// TIA Portal project "Water Control" (V16)

(* hardware
DEVICE "HMI_1"  TP1500 Comfort Portrait
   slot 0: "HMI_1"  TP1500 Comfort Portrait  6AV2 124-0QC02-0AX0  16.0.0.0
   slot 1: "HMI_RT_1"  TP1500 Comfort Portrait  6AV2 124-0QC02-0AX0  16.0.0.0
   slot 5: "HMI_1.IE_CP_1"  PROFINET Interface  16.0.0.0
      slot 1: "PROFINET Interface_1"  PROFINET Interface
         slot 1: "Port_1"  Port
         slot 2: "Port_2"  Port
   slot 6: "HMI_1.IE_CP_2"  PROFINET Interface  16.0.0.0
      slot 1: "PROFINET Interface_GBit"  PROFINET Interface
         slot 1: "Port_1"  Port
   slot 7: "HMI_1.MPI/DP_CP_1"  MPI/DP Interface  16.0.0.0
DEVICE "S71500/ET200MP station_1"  S7-1500 station
   slot 0: "Rail_0"  Rack  6ES7 590-1***0-0AA0
   slot 1: "PLC_1"  CPU 1511-1 PN  6ES7 511-1AK02-0AB0  V2.8
      slot 3: "CPU display_1"  6ES7591-1AA00-0AA0
      slot 32768: "PROFINET interface_1"  X1
         slot 32769: "Port_1"  X1 P1
         slot 32770: "Port_2"  X1 P2
      slot 34817: "Virtual CP interface port_1"  Virtual CP interface port  Virtual CP interface port
*)

// ===== PLC "PLC_1"  CPU 1511-1 PN =====

VAR_GLOBAL   // PLC tag table "Default tag table"
   "Min. Water Level" AT %M0.0 : Bool;
   "Lower Water Level" AT %M0.1 : Bool;
   "Upper Water Level" AT %M0.2 : Bool;
   "Max. Water Level" AT %M0.3 : Bool;
   "Heating" AT %M1.1 : Bool;
   "Inlet Valve Slow" AT %M1.2 : Bool;
   "Inlet Valve Fast" AT %M1.3 : Bool;
   "Oulet Valve" AT %M1.4 : Bool;
   "Water Level" AT %M0.4 : Bool;
   "PTRIG1" AT %M0.5 : Bool;
   "PTRIG2" AT %M0.6 : Bool;
   "PTRIG3" AT %M0.7 : Bool;
   "PTRIG4" AT %M1.0 : Bool;
   "PTRIG5" AT %M1.5 : Bool;
   "Start" AT %M2.0 : Bool;
   "PTRIG6" AT %M1.6 : Bool;
   "Min Sensör arızalı" AT %M1.7 : Bool;
   "RESET" AT %M2.1 : Bool;
END_VAR

DATA_BLOCK "Sıcaklık Bilgileri"   // DB1
{ S7_Optimized_Access := 'TRUE' }
VERSION : 0.1
   VAR
      "Temp. Min Set" : Real;
      "Temp. Max Set" : Real;
      "Temp.Act Value" : Int;
      "Temp Min" : Bool;
      Heating : Bool;
      "Temp Max" : Bool;
   END_VAR
BEGIN
END_DATA_BLOCK

ORGANIZATION_BLOCK "Main"   // OB1, LAD, ProgramCycle
TITLE = "Main Program Sweep (Cycle)"
{ S7_Optimized_Access := 'TRUE' }
VERSION : 0.1
   VAR_INPUT
      Initial_Call : Bool;   // Initial call of this OB
      Remanence : Bool;   // =True, if remanent data are available
   END_VAR
   VAR_TEMP   // added for the SCL form of the ladder/FBD networks
      _w1 : Bool;
      _w2 : Bool;
      _w3 : Bool;
      _w4 : Bool;
      _w5 : Bool;
      _w6 : Bool;
   END_VAR
BEGIN

REGION Network 1: Min Max Temp info
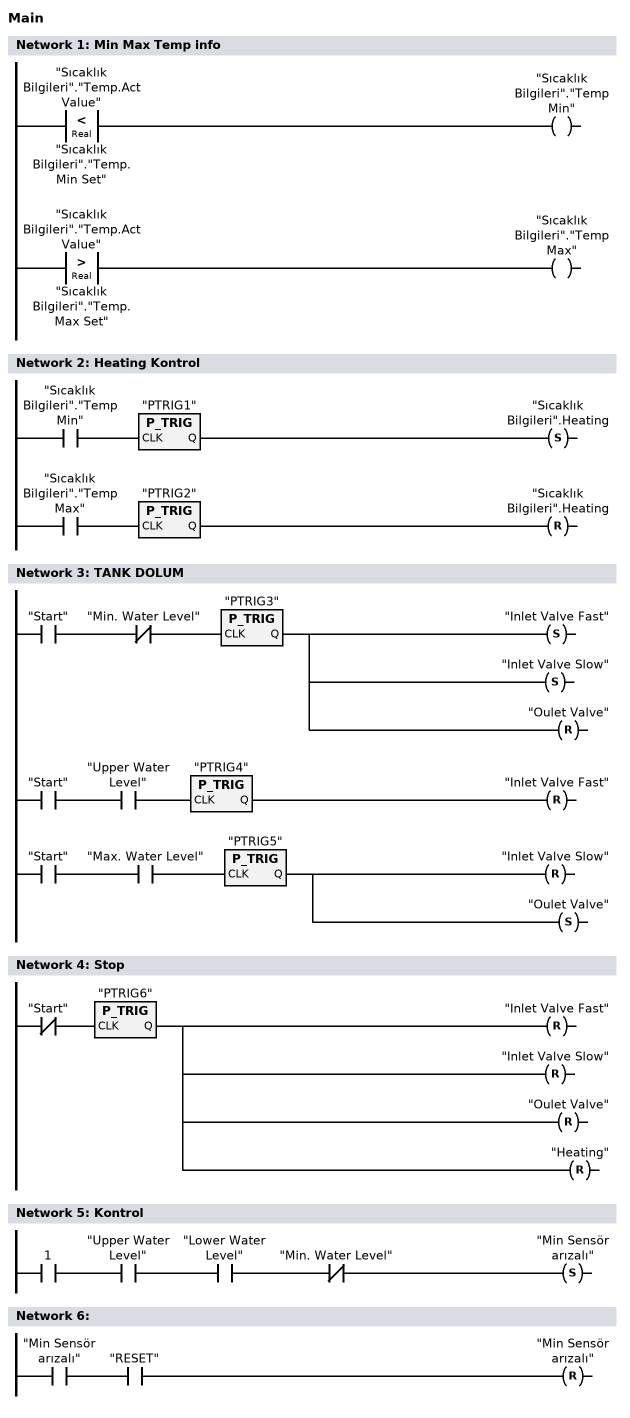
   RUNG wire#powerrail
      { S7_Templates := "SrcType := Real" } LT_Contact(in1 := "Sıcaklık Bilgileri"."Temp.Act Value", in2 := "Sıcaklık Bilgileri"."Temp. Min Set")
      Coil( "Sıcaklık Bilgileri"."Temp Min" )
   END_RUNG
   RUNG wire#powerrail
      { S7_Templates := "SrcType := Real" } GT_Contact(in1 := "Sıcaklık Bilgileri"."Temp.Act Value", in2 := "Sıcaklık Bilgileri"."Temp. Max Set")
      Coil( "Sıcaklık Bilgileri"."Temp Max" )
   END_RUNG
   // the same network as SCL:
   "Sıcaklık Bilgileri"."Temp Min" := "Sıcaklık Bilgileri"."Temp.Act Value" < "Sıcaklık Bilgileri"."Temp. Min Set";
   "Sıcaklık Bilgileri"."Temp Max" := "Sıcaklık Bilgileri"."Temp.Act Value" > "Sıcaklık Bilgileri"."Temp. Max Set";
END_REGION

REGION Network 2: Heating Kontrol
   RUNG wire#powerrail
      Contact( "Sıcaklık Bilgileri"."Temp Min" )
      P_Trig( "PTRIG1" )
      S_Coil( "Sıcaklık Bilgileri".Heating )
   END_RUNG
   RUNG wire#powerrail
      Contact( "Sıcaklık Bilgileri"."Temp Max" )
      P_Trig( "PTRIG2" )
      R_Coil( "Sıcaklık Bilgileri".Heating )
   END_RUNG
   // the same network as SCL:
   #_w1 := "Sıcaklık Bilgileri"."Temp Min" AND NOT "PTRIG1";   // rising edge
   "PTRIG1" := "Sıcaklık Bilgileri"."Temp Min";
   IF #_w1 THEN "Sıcaklık Bilgileri".Heating := TRUE; END_IF;
   #_w2 := "Sıcaklık Bilgileri"."Temp Max" AND NOT "PTRIG2";   // rising edge
   "PTRIG2" := "Sıcaklık Bilgileri"."Temp Max";
   IF #_w2 THEN "Sıcaklık Bilgileri".Heating := FALSE; END_IF;
END_REGION

REGION Network 3: TANK DOLUM
   RUNG wire#powerrail
      Contact( "Start" )
      I_Contact( "Min. Water Level" )
      P_Trig( "PTRIG3" )
      wire#w1
      S_Coil( "Inlet Valve Fast" )
   END_RUNG
   RUNG wire#w1
      S_Coil( "Inlet Valve Slow" )
   END_RUNG
   RUNG wire#w1
      R_Coil( "Oulet Valve" )
   END_RUNG
   RUNG wire#powerrail
      Contact( "Start" )
      Contact( "Upper Water Level" )
      P_Trig( "PTRIG4" )
      R_Coil( "Inlet Valve Fast" )
   END_RUNG
   RUNG wire#powerrail
      Contact( "Start" )
      Contact( "Max. Water Level" )
      P_Trig( "PTRIG5" )
      wire#w2
      R_Coil( "Inlet Valve Slow" )
   END_RUNG
   RUNG wire#w2
      S_Coil( "Oulet Valve" )
   END_RUNG
   // the same network as SCL:
   #_w1 := "Start" AND NOT "Min. Water Level";
   #_w2 := #_w1 AND NOT "PTRIG3";   // rising edge
   "PTRIG3" := #_w1;
   IF #_w2 THEN
       "Inlet Valve Fast" := TRUE;
       "Inlet Valve Slow" := TRUE;
       "Oulet Valve" := FALSE;
   END_IF;
   #_w3 := "Start" AND "Upper Water Level";
   #_w4 := #_w3 AND NOT "PTRIG4";   // rising edge
   "PTRIG4" := #_w3;
   IF #_w4 THEN "Inlet Valve Fast" := FALSE; END_IF;
   #_w5 := "Start" AND "Max. Water Level";
   #_w6 := #_w5 AND NOT "PTRIG5";   // rising edge
   "PTRIG5" := #_w5;
   IF #_w6 THEN
       "Inlet Valve Slow" := FALSE;
       "Oulet Valve" := TRUE;
   END_IF;
END_REGION

REGION Network 4: Stop
   RUNG wire#powerrail
      I_Contact( "Start" )
      P_Trig( "PTRIG6" )
      wire#w1
      R_Coil( "Inlet Valve Fast" )
   END_RUNG
   RUNG wire#w1
      R_Coil( "Inlet Valve Slow" )
   END_RUNG
   RUNG wire#w1
      R_Coil( "Oulet Valve" )
   END_RUNG
   RUNG wire#w1
      R_Coil( "Heating" )
   END_RUNG
   // the same network as SCL:
   #_w1 := NOT "Start" AND NOT "PTRIG6";   // rising edge
   "PTRIG6" := NOT "Start";
   IF #_w1 THEN
       "Inlet Valve Fast" := FALSE;
       "Inlet Valve Slow" := FALSE;
       "Oulet Valve" := FALSE;
       "Heating" := FALSE;
   END_IF;
END_REGION

REGION Network 5: Kontrol
   RUNG wire#powerrail
      Contact( 1 )
      Contact( "Upper Water Level" )
      Contact( "Lower Water Level" )
      I_Contact( "Min. Water Level" )
      S_Coil( "Min Sensör arızalı" )
   END_RUNG
   // the same network as SCL:
   IF 1 AND "Upper Water Level" AND "Lower Water Level" AND NOT "Min. Water Level" THEN
       "Min Sensör arızalı" := TRUE;
   END_IF;
END_REGION

REGION Network 6
   RUNG wire#powerrail
      Contact( "Min Sensör arızalı" )
      Contact( "RESET" )
      R_Coil( "Min Sensör arızalı" )
   END_RUNG
   // the same network as SCL:
   IF "Min Sensör arızalı" AND "RESET" THEN "Min Sensör arızalı" := FALSE; END_IF;
END_REGION
END_ORGANIZATION_BLOCK

(* ===== HMI "HMI_RT_1" =====
system functions are stored by id; their names below are inferred from use
connection "HMI_Connection_3": ETHERNET, S7_1500_OMS

HMI tags "Default tag table"
   "Tag_ScreenNumber" : UInt, internal
   "Sıcaklık Bilgileri_Temp. Min Set" : Real = PLC "Sıcaklık Bilgileri"."Temp. Min Set", 1 s
   "Sıcaklık Bilgileri_Temp. Max Set" : Real = PLC "Sıcaklık Bilgileri"."Temp. Max Set", 1 s
   "Inlet Valve Fast" : Bool = PLC "Inlet Valve Fast" AT %M1.3, 1 s
   "Inlet Valve Slow" : Bool = PLC "Inlet Valve Slow" AT %M1.2, 1 s
   "Oulet Valve" : Bool = PLC "Oulet Valve" AT %M1.4, 1 s
   "Sıcaklık Bilgileri_Temp Min" : Bool = PLC "Sıcaklık Bilgileri"."Temp Min", 1 s
   "Sıcaklık Bilgileri_Temp Max" : Bool = PLC "Sıcaklık Bilgileri"."Temp Max", 1 s
   "Min. Water Level" : Bool = PLC "Min. Water Level" AT %M0.0, 1 s
   "Upper Water Level" : Bool = PLC "Upper Water Level" AT %M0.2, 1 s
   "Max. Water Level" : Bool = PLC "Max. Water Level" AT %M0.3, 1 s
   "Lower Water Level" : Bool = PLC "Lower Water Level" AT %M0.1, 1 s
   "Sıcaklık Bilgileri_Temp.Act Value" : Int = PLC "Sıcaklık Bilgileri"."Temp.Act Value", 1 s
   "Sıcaklık Bilgileri_Heating" : Bool = PLC "Sıcaklık Bilgileri".Heating, 1 s
   "Start" : Bool = PLC Start AT %M2.0, 1 s
   "RESET" : Bool = PLC RESET AT %M2.1, 1 s
   "Min Sensör arızalı" : Bool = PLC "Min Sensör arızalı" AT %M1.7, 1 s

screen "Root screen" 800x1220, template "Template_1"
   on GenerateScreen: SetTag("Tag_ScreenNumber", 1)
   IOField "I/O field_1" at 265,163 size 138x37; FormatPattern 9999.9
      ProcessValue <- "Sıcaklık Bilgileri_Temp. Min Set"
   IOField "I/O field_2" at 265,219 size 138x37; FormatPattern 9999.9
      ProcessValue <- "Sıcaklık Bilgileri_Temp. Max Set"
   TextField "Text field_1" at 79,168 size 180x27; Text 'Min Sıcaklık Set:'
   TextField "Text field_2" at 75,224 size 184x27; Text 'Max Sıcaklık Set:'
   Circle "Circle_1" at 144,320 size 48x48
      Appearance <- "Sıcaklık Bilgileri_Temp Min"
   Circle "Circle_2" at 361,320 size 48x48
      Appearance <- "Sıcaklık Bilgileri_Temp Max"
   TextField "Text field_4" at 102,292 size 131x27; Text 'Min Sıcaklık'
   TextField "Text field_5" at 317,292 size 135x27; Text 'Max Sıcaklık'
   Button "Button_1" at 59,722 size 184x44; TextOff 'Min Water Level'
      on Press: InvertBit("Min. Water Level")
      Appearance <- "Min. Water Level"
   Button "Button_2" at 59,640 size 184x44; TextOff 'Lower Water Level'
      on Press: InvertBit("Lower Water Level")
      Appearance <- "Lower Water Level"
   Button "Button_3" at 59,558 size 184x44; TextOff 'Upper Water Level'
      on Press: InvertBit("Upper Water Level")
      Appearance <- "Upper Water Level"
   Button "Button_4" at 59,476 size 184x44; TextOff 'Max Water Level'
      on Press: InvertBit("Max. Water Level")
      Appearance <- "Max. Water Level"
   Circle "Circle_3" at 564,475 size 48x48
      Appearance <- "Inlet Valve Slow"
   Circle "Circle_4" at 564,557 size 48x48
      Appearance <- "Inlet Valve Fast"
   Circle "Circle_5" at 564,639 size 48x48
      Appearance <- "Oulet Valve"
   TextField "Text field_6" at 416,485 size 114x27; Text 'Inlet Slow'
   TextField "Text field_7" at 416,567 size 107x27; Text 'Inlet Fast'
   TextField "Text field_8" at 416,649 size 127x27; Text 'Oulet Value'
   Circle "Circle_6" at 564,721 size 48x48
      Appearance <- "Sıcaklık Bilgileri_Heating"
   TextField "Text field_9" at 420,731 size 87x27; Text 'Heating'
   Slider "Slider_1" at 541,112 size 132x300; Caption 'Aktüel Sıcaklık'
      ProcessValue <- "Sıcaklık Bilgileri_Temp.Act Value"
   Button "Button_5" at 240,17 size 323x64; TextOff 'Start'; TextOn 'Stop'
      Appearance <- "Start"
      on Press: InvertBit("Start")
   Button "Button_6" at 59,809 size 185x32; TextOff 'ARIZA RESET'
      Appearance <- "RESET"
      on Press: function_b14e0dd5("RESET", 0)
   TextField "Text field_3" at 420,818 size 176x25; Text 'Min Sensör Arızalı'
      Visibility <- "Min Sensör arızalı"

Template "Template_1" 800x1220
   Button "Exit" at 720,1159 size 78x59; TextOff 'Exit'; PictureOff "ExitRuntime_TP1500_Comfort_Portrait_TR"; PictureOn "ExitRuntime_TP1500_Comfort_Portrait_TR"
      on Release: StopRuntime(0)
   Button "Template_Button" at 640,1159 size 78x59; TextOff 'Text'
   Button "Template_Button_1" at 560,1159 size 78x59; TextOff 'Text'
   Button "Template_Button_2" at 480,1159 size 78x59; TextOff 'Text'
   Button "Template_Button_3" at 400,1159 size 78x59; TextOff 'Text'
   Button "Template_Button_4" at 321,1159 size 78x59; TextOff 'Text'
   Button "Template_Button_5" at 241,1159 size 78x59; TextOff 'Text'
   Button "Template_Button_6" at 161,1159 size 78x59; TextOff 'Text'
   Button "Alarms" at 81,1159 size 78x59; TextOff 'Alarms'; PictureOff "AlarmDisplay_TP1500_Comfort_Portrait_TR"; PictureOn "AlarmDisplay_TP1500_Comfort_Portrait_TR"
      on Release: function_ef3f5d25("Alarm window_Unacknowledged", -1)
   Button "Start screen" at 1,1159 size 78x59; TextOff 'Start screen'; PictureOff "NavigateHome_TP1500_Comfort_Portrait_TR"; PictureOn "NavigateHome_TP1500_Comfort_Portrait_TR"
      on Release: ActivateScreen("Root screen", 0)
*)